FUNCTION_BLOCK CmdValvePump (* CAT Function Block Type *)
  (* Standard: 61499-2 *)
  (* Version 0.0, 6/7/2026, Schneider Electric, template *)
  PACKAGE SE.Nereda;
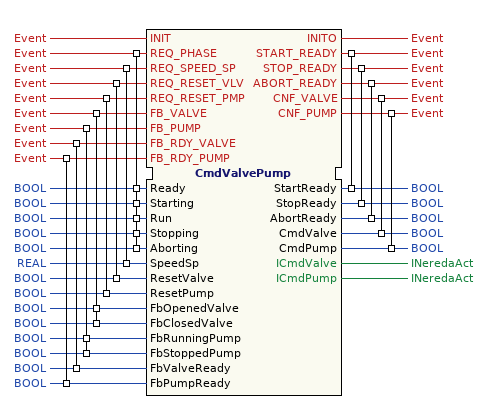
  EVENT_INPUT
    INIT;
    REQ_PHASE WITH Ready, Starting, Run, Stopping, Aborting;
    REQ_SPEED_SP WITH SpeedSp;
    REQ_RESET_VLV WITH ResetValve;
    REQ_RESET_PMP WITH ResetPump;
    FB_VALVE WITH FbOpenedValve, FbClosedValve;
    FB_PUMP WITH FbRunningPump, FbStoppedPump;
    FB_RDY_VALVE WITH FbValveReady;
    FB_RDY_PUMP WITH FbPumpReady;
  END_EVENT
  EVENT_OUTPUT
    INITO;
    START_READY WITH StartReady;
    STOP_READY WITH StopReady;
    ABORT_READY WITH AbortReady;
    CNF_VALVE WITH CmdValve;
    CNF_PUMP WITH CmdPump;
  END_EVENT
  VAR_INPUT
    Ready : BOOL;
    Starting : BOOL;
    Run : BOOL;
    Stopping : BOOL;
    Aborting : BOOL;
    SpeedSp : REAL;
    ResetValve : BOOL;
    ResetPump : BOOL;
    FbOpenedValve : BOOL;
    FbClosedValve : BOOL;
    FbRunningPump : BOOL;
    FbStoppedPump : BOOL;
    FbValveReady : BOOL;
    FbPumpReady : BOOL;
  END_VAR
  VAR_OUTPUT
    StartReady : BOOL;
    StopReady : BOOL;
    AbortReady : BOOL;
    CmdValve : BOOL;
    CmdPump : BOOL;
  END_VAR
  PLUGS
    ICmdValve : INeredaAct;
    ICmdPump : INeredaAct;
  END_PLUGS
  (* 01 - FUNCTIONNAL INPUT INTERFACE *)
  (* 00 - INITIALIZATION *)
  (* 05 - LOGIC *)
  (* 06 - HMI INTERFACE *)
  (* 03 - FIELD INTERFACE *)
  (* 02 - FUNCTIONNAL OUTPUT INTERFACE *)
  (* Command Logic *)
  FBS
    CmdLogic : CmdValvePumpBasic;
    IThis : CmdValvePump_HMI(QI := TRUE);
    ValveCmdSmooth : boolValueChanged;
    PumpCmdSmooth : boolValueChanged;
    FbOpenValve : DS_SELECTX_2536758B411A6CE51; {SET_ATTRIBUTE(Configuration.GenericFBType.InterfaceParams, Runtime.Standard#CNTX:=2;CNTY:=1;DI${CNTX,_,CNTY$}:BOOL)}
    FbCloseValve : DS_SELECTX_2536758B411A6CE51; {SET_ATTRIBUTE(Configuration.GenericFBType.InterfaceParams, Runtime.Standard#CNTX:=2;CNTY:=1;DI${CNTX,_,CNTY$}:BOOL)}
    FbRunPump : DS_SELECTX_2536758B411A6CE51; {SET_ATTRIBUTE(Configuration.GenericFBType.InterfaceParams, Runtime.Standard#CNTX:=2;CNTY:=1;DI${CNTX,_,CNTY$}:BOOL)}
    FbStopPump : DS_SELECTX_2536758B411A6CE51; {SET_ATTRIBUTE(Configuration.GenericFBType.InterfaceParams, Runtime.Standard#CNTX:=2;CNTY:=1;DI${CNTX,_,CNTY$}:BOOL)}
    FbReadyPump : DS_SELECTX_2536758B411A6CE51; {SET_ATTRIBUTE(Configuration.GenericFBType.InterfaceParams, Runtime.Standard#CNTX:=2;CNTY:=1;DI${CNTX,_,CNTY$}:BOOL)}
    FbReadyValve : DS_SELECTX_2536758B411A6CE51; {SET_ATTRIBUTE(Configuration.GenericFBType.InterfaceParams, Runtime.Standard#CNTX:=2;CNTY:=1;DI${CNTX,_,CNTY$}:BOOL)}
    ValveCmd : BOOL2INT;
    PumpCmd : BOOL2INT;
  END_FBS
  EVENT_CONNECTIONS
    INIT TO IThis.C65860F65D546C3D;
    IThis.C4541B09DE1DCFD1 TO INITO;
    ValveCmdSmooth.CHD TO CNF_VALVE;
    PumpCmdSmooth.CHD TO CNF_PUMP;
    FB_VALVE TO FbOpenValve.REQ2;
    FbOpenValve.CNF1 TO FbCloseValve.REQ1;
    FbOpenValve.CNF2 TO FbCloseValve.REQ2;
    FbRunPump.CNF1 TO FbStopPump.REQ1;
    FbRunPump.CNF2 TO FbStopPump.REQ2;
    FB_PUMP TO FbRunPump.REQ2;
    FB_RDY_VALVE TO FbReadyValve.REQ2;
    FB_RDY_PUMP TO FbReadyPump.REQ2;
    REQ_PHASE TO CmdLogic.READY;
    REQ_PHASE TO CmdLogic.STARTING;
    REQ_PHASE TO CmdLogic.RUN;
    REQ_PHASE TO CmdLogic.STOPPING;
    REQ_PHASE TO CmdLogic.ABORTING;
    REQ_SPEED_SP TO ICmdPump.1E00729184986247;
    REQ_RESET_VLV TO ICmdValve.37BBC1F841739733;
    REQ_RESET_PMP TO ICmdPump.37BBC1F841739733;
    CmdLogic.001688431DB935DE TO IThis.7FB6E91A6128B6A3;
    FbCloseValve.IND TO CmdLogic.VALVE_FB_OPEN;
    FbStopPump.IND TO CmdLogic.PUMP_FB_RUN;
    FbReadyValve.IND TO CmdLogic.VALVE_AVAILABLE;
    FbReadyPump.IND TO CmdLogic.PUMP_NO_AVAILABLE;
    CmdLogic.VALVE_CNF TO ValveCmdSmooth.REQ;
    ValveCmdSmooth.CHD TO ValveCmd.DD5870AA881150BB;
    PumpCmdSmooth.CHD TO PumpCmd.DD5870AA881150BB;
    CmdLogic.PUMP_CNF TO PumpCmdSmooth.REQ;
    CmdLogic.START_READY TO START_READY;
    CmdLogic.STOP_READY TO STOP_READY;
    CmdLogic.ABORTED_READY TO ABORT_READY;
    ICmdValve.9CD053F8408797ED TO FbOpenValve.REQ1;
    ICmdValve.CC753684FA882790 TO FbReadyValve.REQ1;
    ICmdPump.9CD053F8408797ED TO FbRunPump.REQ1;
    ICmdPump.CC753684FA882790 TO FbReadyPump.REQ1;
    ValveCmd.6FC99A5BD1C38561 TO ICmdValve.0F1CDF9A9B4A227A;
    PumpCmd.6FC99A5BD1C38561 TO ICmdPump.0F1CDF9A9B4A227A;
  END_CONNECTIONS
  DATA_CONNECTIONS
    ValveCmdSmooth.Output TO CmdValve;
    PumpCmdSmooth.Output TO CmdPump;
    FbOpenedValve TO FbOpenValve.DI2_1;
    FbClosedValve TO FbCloseValve.DI2_1;
    FbRunningPump TO FbRunPump.DI2_1;
    FbStoppedPump TO FbStopPump.DI2_1;
    FbValveReady TO FbReadyValve.DI2_1;
    FbPumpReady TO FbReadyPump.DI2_1;
    Ready TO CmdLogic.Ready;
    Starting TO CmdLogic.Starting;
    Run TO CmdLogic.RunningState;
    Stopping TO CmdLogic.Stopping;
    Aborting TO CmdLogic.Aborting;
    SpeedSp TO ICmdPump.1BC103921BBFDA0B;
    ResetValve TO ICmdValve.EA28053F07575F36;
    ResetPump TO ICmdPump.EA28053F07575F36;
    CmdLogic.DB4AE032AE08C110 TO IThis.67D1364BABA62FC3;
    ValveCmdSmooth.Output TO ValveCmd.4573FC8F228EB71D;
    PumpCmdSmooth.Output TO PumpCmd.4573FC8F228EB71D;
    CmdLogic.Valve TO ValveCmdSmooth.Input;
    CmdLogic.Pump TO PumpCmdSmooth.Input;
    CmdLogic.StartReady TO StartReady;
    CmdLogic.StopReady TO StopReady;
    CmdLogic.AbortedReady TO AbortReady;
    FbOpenValve.OUT1 TO CmdLogic.ValveFbOpen;
    FbCloseValve.OUT1 TO CmdLogic.ValveFbClose;
    FbRunPump.OUT1 TO CmdLogic.PumpFbRunning;
    FbStopPump.OUT1 TO CmdLogic.PumpFbStopped;
    FbReadyValve.OUT1 TO CmdLogic.ValveAvailable;
    FbReadyPump.OUT1 TO CmdLogic.PumpNotAvailable;
    ICmdValve.7F6CC7FEB9223DF3 TO FbOpenValve.DI1_1;
    ICmdValve.A8D6C4A1FDCCA991 TO FbCloseValve.DI1_1;
    ICmdValve.8A8A07EFCDA1443C TO FbReadyValve.DI1_1;
    ICmdPump.D83B5BDEFA4D797C TO FbStopPump.DI1_1;
    ICmdPump.B762734C094A7162 TO FbRunPump.DI1_1;
    ICmdPump.8A8A07EFCDA1443C TO FbReadyPump.DI1_1;
    ValveCmd.A6DEF5F9C27C1848 TO ICmdValve.710D7FC54EE3F35A;
    PumpCmd.A6DEF5F9C27C1848 TO ICmdPump.710D7FC54EE3F35A;
  END_CONNECTIONS
END_FUNCTION_BLOCK
